(* PLC project PLC1, Beckhoff Automation GmbH TwinCAT PLC Control 3.5.13.21 *)
(* stored: creationDateTime 2023-01-20T09:34:25.9600499, modificationDateTime 2023-01-20T09:34:25.9600499 *)

FUNCTION_BLOCK FB_SafetyBckpRstr
  VAR
    _fbSaveLogicProgram : FB_SAVELOGICPROGRAM;
    _fbRestoreLogicProgram : FB_RESTORELOGICPROGRAM;
    refEcNetId : REFERENCE TO ARRAY [0..5] OF BYTE;
    refBuffer : REFERENCE TO ARRAY [0..16#FFFF] OF BYTE;
    nEcPort : WORD;
    sFileName : T_MaxString;
    sNetIdRWFile : T_AmsNetID;
  END_VAR

            
          

METHOD RestoreLogicProgram : BOOL
  VAR_INPUT
    bExecute : BOOL;
  END_VAR
  VAR_OUTPUT
    stTcOutputsSafetyRstr : ST_TcOutputsSafetyBckpRstr;
  END_VAR
                  IF __ISVALIDREF(refBuffer) AND __ISVALIDREF(refEcNetId) THEN
_fbRestoreLogicProgram(
	bExecute:= bExecute, 
	au8EcatNetId:= refEcNetId, 
	u16EcatPort:= nEcPort, 
	u32BufferAddress:= ADR(refBuffer), 
	u32BufferSize:= SIZEOF(refBuffer), 
	sFileName:= sFileName, 
	sNetIDReadFile:= sNetIdRWFile, 
	Done=> stTcOutputsSafetyRstr.stTcGeneralOutputs.bDone, 
	sResult=> stTcOutputsSafetyRstr.sResult, 
	bErr=> stTcOutputsSafetyRstr.stTcGeneralOutputs.bError);	
END_IF

                
END_METHOD

METHOD SaveLogicProgram : BOOL
  VAR_INPUT
    bExecute : BOOL;
  END_VAR
  VAR_OUTPUT
    stTcOutputsSafetyBckp : ST_TcOutputsSafetyBckpRstr;
  END_VAR
                  IF __ISVALIDREF(refBuffer) AND __ISVALIDREF(refEcNetId) THEN
_fbSaveLogicProgram(
	bExecute:= bExecute, 
	au8EcatNetId:= refEcNetId, 
	u16EcatPort:= nEcPort, 
	u32BufferAddress:= ADR(refBuffer) ,
	u32BufferSize:= SIZEOF(refBuffer),  
	sFileName:= sFileName, 
	sNetIDWriteFile:= sNetIdRWFile, 
	Done=> stTcOutputsSafetyBckp.stTcGeneralOutputs.bDone, 
	sResult=> stTcOutputsSafetyBckp.sResult, 
	bErr=> stTcOutputsSafetyBckp.stTcGeneralOutputs.bError);
END_IF



                
END_METHOD

PROPERTY Buffer : REFERENCE TO ARRAY [0..16#FFFF] OF BYTE
SET
                    refBuffer REF= Buffer;
                  
END_SET
END_PROPERTY

PROPERTY EcNetId : REFERENCE TO ARRAY [0..5] OF BYTE
SET
                    refEcNetId REF= EcNetId;
                  
END_SET
END_PROPERTY

PROPERTY EcPort : WORD
SET
                    nEcPort := EcPort;
                  
END_SET
END_PROPERTY

PROPERTY FileName : T_MaxString
GET
                    
                  
END_GET
SET
                    sFileName := FileName;
                  
END_SET
END_PROPERTY

PROPERTY NetIdRWFile : T_AmsNetID
GET
                    
                  
END_GET
SET
                    sNetIdRWFile := NetIdRWFile;
                  
END_SET
END_PROPERTY
END_FUNCTION_BLOCK
